FUNCTION_BLOCK AxesMoveVelocityProcess EXTENDS BaseProcess
VAR_INPUT
	///Arguments to be set, before writing do_request TRUE
	{attribute 'OPC.UA.DA' := '1'}
	set: AxesMoveVelocityProcessArgs;
END_VAR
VAR_OUTPUT
	///Arguments in use by the process, if do_request was accepted
	{attribute 'OPC.UA.DA' := '1'}
	{attribute 'OPC.UA.DA.Access' := '1'}
	get: AxesMoveVelocityProcessArgs;
END_VAR
VAR_IN_OUT
END_VAR
VAR
END_VAR

IF do_request THEN
    do_request_result := request(
    units := set.units,
    value := set.value);
    do_request := FALSE;
END_IF;
SUPER^();

{attribute 'TcRpcEnable' := '1'}
METHOD request : RequestResults
VAR_INPUT
	///Units of the 'value' argument (RADIANS_PER_SECOND, DEGREES_PER_SECOND, ...)
	units: AxesMoveVelocityUnits;
	///Move the axis with this velocity (which units depends on the 'units' argument)
	value: LREAL;
END_VAR
VAR_OUTPUT
END_VAR
VAR_IN_OUT
END_VAR
VAR
END_VAR
IF THIS^.statuses.enabledStatus.enabled THEN
    THIS^.start(
        units := units,
        value := value);
    request := RequestResults.ACCEPTED;
ELSE
    request := RequestResults.REJECTED;
END_IF;
END_METHOD

{attribute 'TcRpcEnable' := '1'}
METHOD start
VAR_INPUT
	///Units of the 'value' argument (RADIANS_PER_SECOND, DEGREES_PER_SECOND, ...)
	units: AxesMoveVelocityUnits;
	///Move the axis with this velocity (which units depends on the 'units' argument)
	value: LREAL;
END_VAR
VAR_OUTPUT
END_VAR
VAR_IN_OUT
END_VAR
VAR
END_VAR
THIS^.get.units := units;
THIS^.get.value := value;
THIS^.statuses.busyStatus( isBusy := TRUE );
THIS^.statuses.healthStatus( isGood := TRUE );
END_METHOD

END_FUNCTION_BLOCK

(* stored: Version 1.1.0.1, ProductVersion 3.1.4019.2
   POU AxesMoveVelocityProcess: Id {d1f1667b-01bf-493a-b7d8-3e1ef0a64230}, SpecialFunc None
   Method request: Id {74b441f6-d40e-4aec-858a-8f841ccb4701}
   Method start: Id {d5662904-73bb-4609-beab-6ca249104144} *)
